INTERFACE I_EnergySource

METHOD GetPower : REAL
END_METHOD

END_INTERFACE

(* stored: Version 1.1.0.1, ProductVersion 3.1.4024.16
   Itf I_EnergySource: Id {10273e1d-355d-4617-9c31-4122d6ff8f46}
   Method GetPower: Id {b63b09d9-2a56-4da4-84a9-9ffccea2cad7} *)
